(* CoDeSys 2.3 library: TestLib.lib *)

(* Data type *)
TYPE eTest :
(
	banana := 1,
	chili := 2,
	apple := 3
);
END_TYPE

(* POU F_Process, ST *)
FUNCTION F_Process : BOOL
VAR_INPUT
END_VAR
VAR
END_VAR
;
END_FUNCTION

(* POU F_TestFunction, ST *)
FUNCTION F_TestFunction : BOOL
VAR_INPUT
	xInput:		BOOL;
END_VAR
VAR
END_VAR
;
END_FUNCTION

(* POU Fb_TestFunctionBlock, ST *)
FUNCTION_BLOCK Fb_TestFunctionBlock
VAR_INPUT
	xInVar:			BOOL;
	rInVar:			REAL;
	wInVar:			WORD;
END_VAR
VAR_OUTPUT
	xOutVar:		BOOL;
	rOutVar:		REAL;
END_VAR
VAR
END_VAR
;
END_FUNCTION_BLOCK
